// TIA Portal project "WM" (V16)

(* hardware
DEVICE "S7-1200 station_1"  S7-1200 Station
   slot 0: "Rack_0"  S7-1200 Rack  Rack  V1.0
   slot 1: "PLC_1"  CPU 1212C AC/DC/Rly  6ES7 212-1BE40-0XB0  V4.4
*)

// ===== PLC "PLC_1"  CPU 1212C AC/DC/Rly =====

VAR_GLOBAL   // PLC tag table "Default tag table"
   "START" AT %I0.1 : Bool;
   "STOP" AT %I0.2 : Bool;
   "MOTOR1" AT %Q0.0 : Bool;
   "MOTOR2" AT %Q0.1 : Bool;
   "TM1" AT %M0.0 : Bool;
   "TM2" AT %M0.1 : Bool;
   "SAVE" AT %M0.2 : Bool;
   "T1ON" AT %M0.3 : Bool;
   "X" AT %M0.4 : Bool;
END_VAR

// folder: System blocks/Program resources

DATA_BLOCK "TIMER1"   // DB1
{ S7_Optimized_Access := 'TRUE' }
AUTHOR : Simatic
FAMILY : IEC
NAME : IEC_TMR
VERSION : 1.0
// stored: InstanceOfName IEC_TIMER
"IEC_TIMER"
BEGIN
END_DATA_BLOCK

DATA_BLOCK "TIMER2"   // DB2
{ S7_Optimized_Access := 'TRUE' }
AUTHOR : Simatic
FAMILY : IEC
NAME : IEC_TMR
VERSION : 1.0
// stored: InstanceOfName IEC_TIMER
"IEC_TIMER"
BEGIN
END_DATA_BLOCK

// folder: (top level)

ORGANIZATION_BLOCK "Main"   // OB1, LAD, ProgramCycle
TITLE = "Main Program Sweep (Cycle)"
{ S7_Optimized_Access := 'TRUE' }
VERSION : 0.1
   VAR_INPUT
      Initial_Call : Bool;   // Initial call of this OB
      Remanence : Bool;   // =True, if remanent data are available
   END_VAR
BEGIN

REGION Network 1
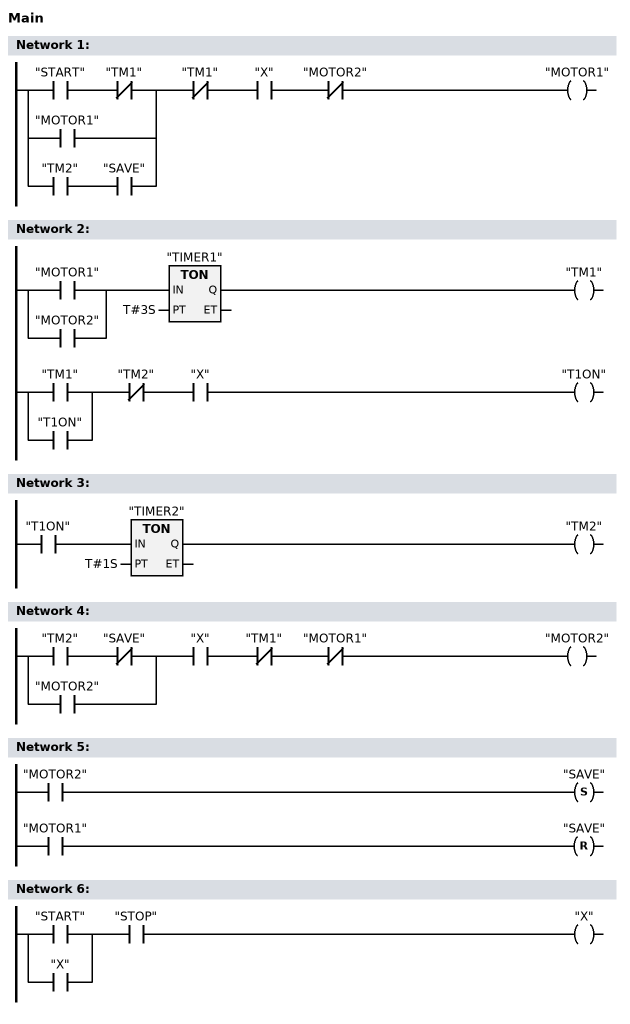
   RUNG wire#powerrail
      Contact( "START" )
      I_Contact( "TM1" )
      wire#w1
      I_Contact( "TM1" )
      Contact( "X" )
      I_Contact( "MOTOR2" )
      Coil( "MOTOR1" )
   END_RUNG
   RUNG wire#powerrail
      Contact( "MOTOR1" )
   END_RUNG wire#w1
   RUNG wire#powerrail
      Contact( "TM2" )
      Contact( "SAVE" )
   END_RUNG wire#w1
   // the same network as SCL:
   "MOTOR1" := (("START" AND NOT "TM1") OR "MOTOR1" OR ("TM2" AND "SAVE")) AND NOT "TM1" AND "X" AND NOT "MOTOR2";
END_REGION

REGION Network 2
   "TIMER1".TON(IN := "MOTOR1" OR "MOTOR2", PT := T#3S);
   "TM1" := "TIMER1".Q;
   "T1ON" := ("TM1" OR "T1ON") AND NOT "TM2" AND "X";
END_REGION

REGION Network 3
   "TIMER2".TON(IN := "T1ON", PT := T#1S);
   "TM2" := "TIMER2".Q;
END_REGION

REGION Network 4
   RUNG wire#powerrail
      Contact( "TM2" )
      I_Contact( "SAVE" )
      wire#w1
      Contact( "X" )
      I_Contact( "TM1" )
      I_Contact( "MOTOR1" )
      Coil( "MOTOR2" )
   END_RUNG
   RUNG wire#powerrail
      Contact( "MOTOR2" )
   END_RUNG wire#w1
   // the same network as SCL:
   "MOTOR2" := (("TM2" AND NOT "SAVE") OR "MOTOR2") AND "X" AND NOT "TM1" AND NOT "MOTOR1";
END_REGION

REGION Network 5
   RUNG wire#powerrail
      Contact( "MOTOR2" )
      S_Coil( "SAVE" )
   END_RUNG
   RUNG wire#powerrail
      Contact( "MOTOR1" )
      R_Coil( "SAVE" )
   END_RUNG
   // the same network as SCL:
   IF "MOTOR2" THEN "SAVE" := TRUE; END_IF;
   IF "MOTOR1" THEN "SAVE" := FALSE; END_IF;
END_REGION

REGION Network 6
   RUNG wire#powerrail
      Contact( "START" )
      wire#w1
      Contact( "STOP" )
      Coil( "X" )
   END_RUNG
   RUNG wire#powerrail
      Contact( "X" )
   END_RUNG wire#w1
   // the same network as SCL:
   "X" := ("START" OR "X") AND "STOP";
END_REGION
END_ORGANIZATION_BLOCK